{attribute 'qualified_only'}
VAR_GLOBAL
	Analog_Inputs_Res AT %I* : ARRAY[1..2] OF INT;
	Analog_Inputs_Res_Values : ARRAY[1..2] OF REAL;
END_VAR

(* stored: Version 1.1.0.1, ProductVersion 3.1.4024.12
   GVL GVL: Id {e63236d2-f5ad-46d7-97fc-ec6caeea6e66} *)
